(* PLC project Gen3Safety, BrAutomation SafeDESIGNER  5.19.0.0 *)
(* stored: companyURL http://www.br-automation.com, creationDateTime Mon Apr 29 14:05:33 2024 *)

PROGRAM Main
  VAR  (* added by the conversion: wires and edge detectors of the diagram *)
    _NOT_S160_OUT : ANY;
    _NOT_S167_OUT : ANY;
    _AND_S92_OUT : ANY;
  END_VAR

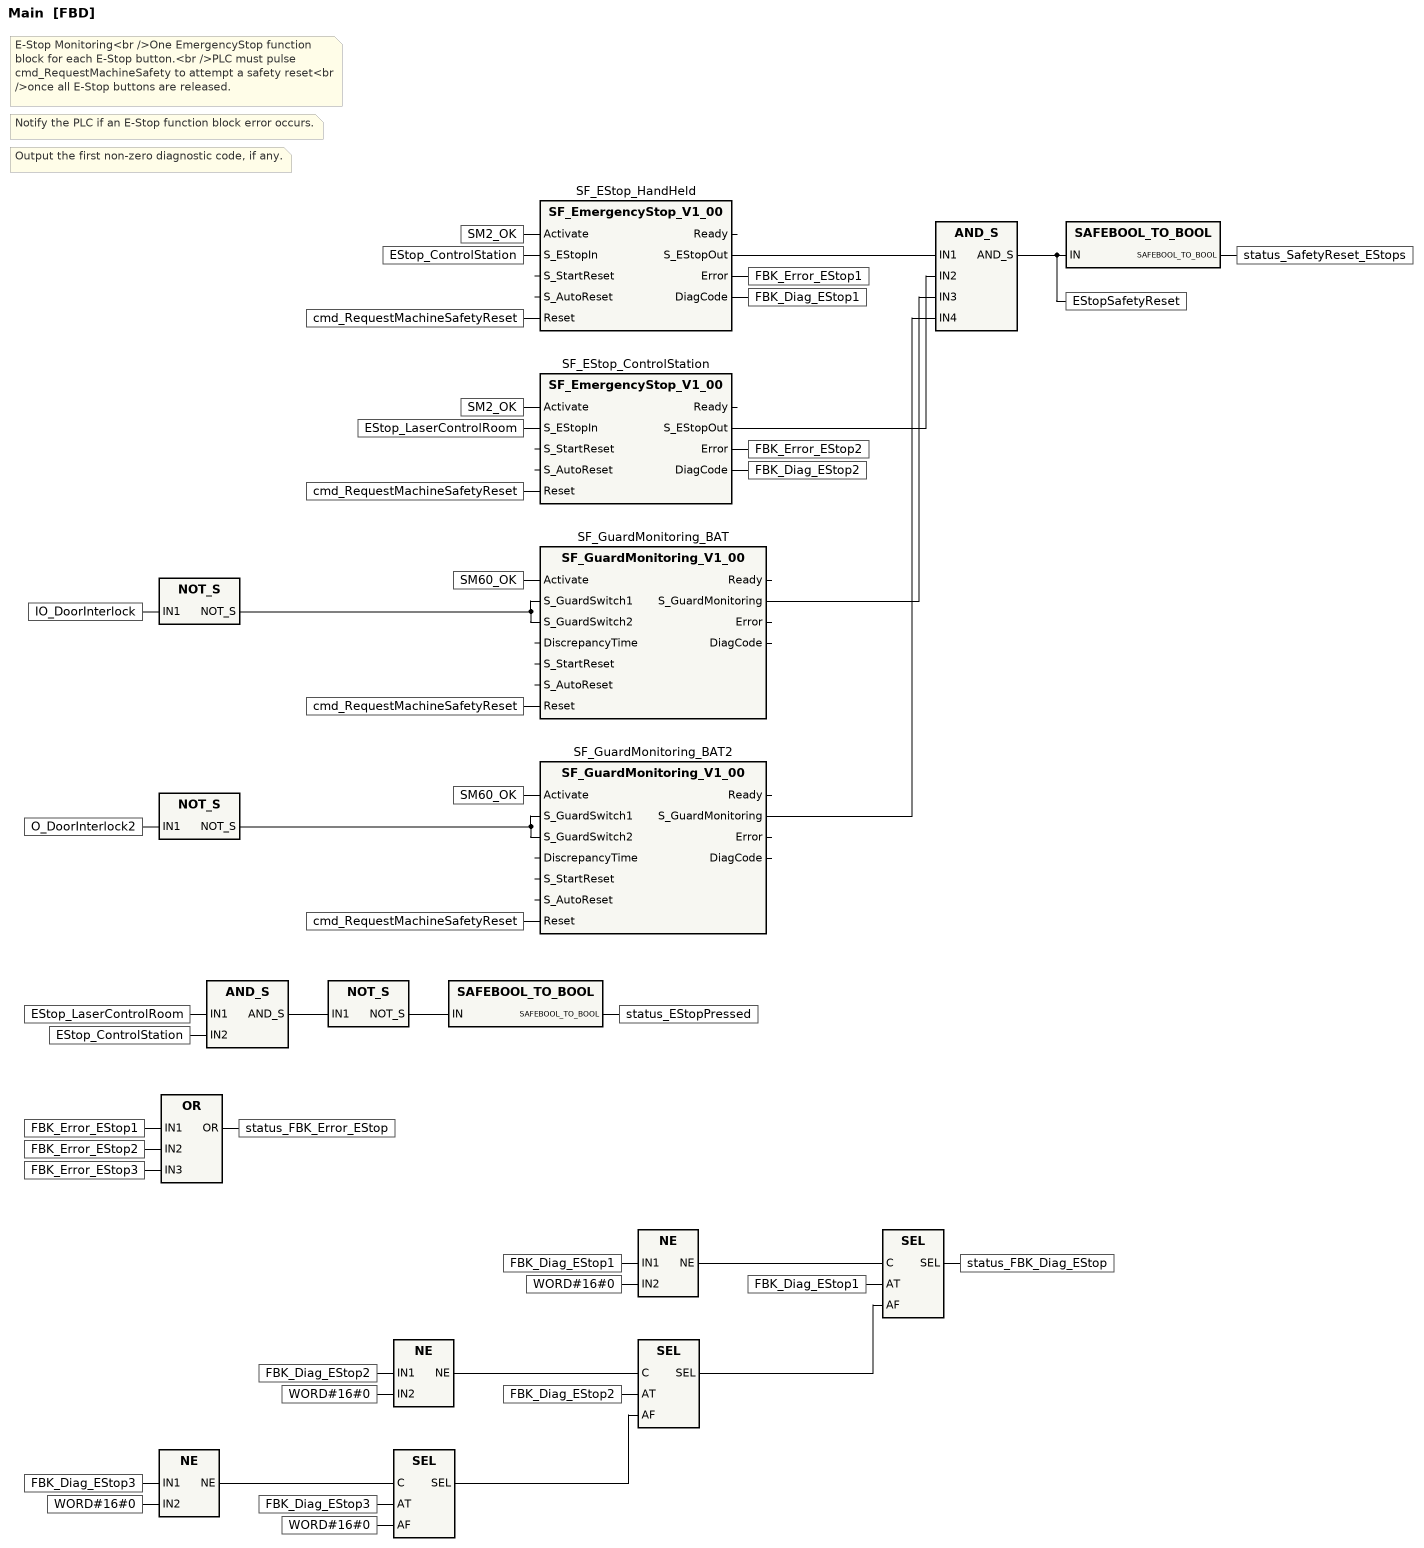
(* FBD diagram, written out as Structured Text *)
(* E-Stop Monitoring<br />One EmergencyStop function block for each E-Stop button.<br />PLC must pulse cmd_RequestMachineSafety to attempt a safety reset<br />once all E-Stop buttons are released. *)
SF_EStop_HandHeld(Activate := SM2_OK, S_EStopIn := EStop_ControlStation, Reset := cmd_RequestMachineSafetyReset);
FBK_Error_EStop1 := SF_EStop_HandHeld.Error;
FBK_Diag_EStop1 := SF_EStop_HandHeld.DiagCode;
SF_EStop_ControlStation(Activate := SM2_OK, S_EStopIn := EStop_LaserControlRoom, Reset := cmd_RequestMachineSafetyReset);
_NOT_S160_OUT := NOT_S(IO_DoorInterlock);
SF_GuardMonitoring_BAT(Activate := SM60_OK, S_GuardSwitch1 := _NOT_S160_OUT, S_GuardSwitch2 := _NOT_S160_OUT, Reset := cmd_RequestMachineSafetyReset);
_NOT_S167_OUT := NOT_S(O_DoorInterlock2);
SF_GuardMonitoring_BAT2(Activate := SM60_OK, S_GuardSwitch1 := _NOT_S167_OUT, S_GuardSwitch2 := _NOT_S167_OUT, Reset := cmd_RequestMachineSafetyReset);
_AND_S92_OUT := AND_S(SF_EStop_HandHeld.S_EStopOut, SF_EStop_ControlStation.S_EStopOut, SF_GuardMonitoring_BAT.S_GuardMonitoring, SF_GuardMonitoring_BAT2.S_GuardMonitoring);
EStopSafetyReset := _AND_S92_OUT;
status_SafetyReset_EStops := SAFEBOOL_TO_BOOL(_AND_S92_OUT);
FBK_Error_EStop2 := SF_EStop_ControlStation.Error;
FBK_Diag_EStop2 := SF_EStop_ControlStation.DiagCode;
status_EStopPressed := SAFEBOOL_TO_BOOL(NOT_S(AND_S(EStop_LaserControlRoom, EStop_ControlStation)));
(* Notify the PLC if an E-Stop function block error occurs. *)
status_FBK_Error_EStop := FBK_Error_EStop1 OR FBK_Error_EStop2 OR FBK_Error_EStop3;
(* Output the first non-zero diagnostic code, if any. *)
status_FBK_Diag_EStop := SEL(FBK_Diag_EStop1 <> WORD#16#0, FBK_Diag_EStop1, SEL(FBK_Diag_EStop2 <> WORD#16#0, FBK_Diag_EStop2, SEL(FBK_Diag_EStop3 <> WORD#16#0, FBK_Diag_EStop3, WORD#16#0)));
END_PROGRAM
